FUNCTION_BLOCK ASR_SR_TO_2EVENTS (* Composite FB for convert ASR to 2 EVENTS *)
  (* Standard: 61499-2; Description: Copyright (c) 2024 HR Agrartechnik GmbH This program and the accompanying materials are made available under the terms of the Eclipse Public License 2.0 which is available at https://www.eclipse.org/legal/epl-2.0/ SPDX-License-Identifier: EPL-2.0 *)
  (* Version 1.0, 2024-04-24, Franz Höpfinger, HR Agrartechnik GmbH *)
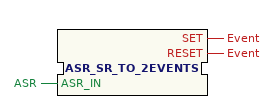
  EVENT_OUTPUT
    SET; (* Set / Switch on *)
    RESET; (* Reset / Switch off *)
  END_EVENT
  SOCKETS
    ASR_IN : ASR; (* Adapter Input *)
  END_SOCKETS
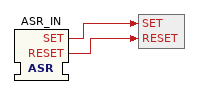
  EVENT_CONNECTIONS
    ASR_IN.SET TO SET;
    ASR_IN.RESET TO RESET;
  END_CONNECTIONS
END_FUNCTION_BLOCK
